FUNCTION_BLOCK FB_LeakTest
VAR_INPUT
    bExecute       		: BOOL;  		// Starts the leak test
    eSolenoidPosition 	: E_SolenoidSet;// Defines the solenoid valve positions
    tMonitorTime   		: TIME;  		// Monitoring time duration
    rPressureLimit 		: REAL;  		// Minimum required pressure limit
END_VAR

VAR_OUTPUT
    bLeakTestDone  : BOOL;  		// Indicates if the test was successful
    bLeakTestError : BOOL;  		// Indicates if an error occurred during the test
    sLTMessageError: STRING(100);  	// Error message describing the failure
END_VAR

VAR
    fbValveControl1 	: FB_ValvePositionControl;
    fbValveControl2 	: FB_ValvePositionControl;
    fbValveControl3 	: FB_ValvePositionControl;
    fbValveControl4 	: FB_ValvePositionControl;
    fbValveControl5 	: FB_ValvePositionControl;
    fbSolenoidControl 	: FB_SolenoidControl;
    fbSensorScale   	: FB_SensorScaling;
    tStartTime      	: TIME;
    rScaledPressure 	: REAL;
    eState          	: (IDLE, POSITION_VALVES, SET_SOLENOIDS, PRESSURIZE, MONITOR, DONE, ERROR);
END_VAR

CASE eState OF
    IDLE:
        // Waits for the execution command to start the test
        IF bExecute THEN
            eState := POSITION_VALVES;
        END_IF;

    POSITION_VALVES:
        // Moves all 6-position valves to position 5
        fbValveControl1(bEnable := TRUE, iValvePosition := 5, ServoAxis := GVL_Motion.M4Valve1.Axis);
        fbValveControl2(bEnable := TRUE, iValvePosition := 5, ServoAxis := GVL_Motion.M5Valve2.Axis);
        fbValveControl3(bEnable := TRUE, iValvePosition := 5, ServoAxis := GVL_Motion.M6Valve3.Axis);
        fbValveControl4(bEnable := TRUE, iValvePosition := 5, ServoAxis := GVL_Motion.M7Valve4.Axis);
        fbValveControl5(bEnable := TRUE, iValvePosition := 5, ServoAxis := GVL_Motion.M8Valve5.Axis);
        
        // If all valves have moved successfully, proceed to setting solenoids
        IF fbValveControl1.bMoveDone AND fbValveControl2.bMoveDone AND fbValveControl3.bMoveDone AND fbValveControl4.bMoveDone AND fbValveControl5.bMoveDone THEN
            eState := SET_SOLENOIDS;
        // If any valve encounters an error, transition to ERROR state
        ELSIF fbValveControl1.bError OR fbValveControl2.bError OR fbValveControl3.bError OR fbValveControl4.bError OR fbValveControl5.bError THEN
            bLeakTestError := TRUE;
            sLTMessageError := 'Failed to position valves';
            eState := ERROR;
        END_IF;
    
    SET_SOLENOIDS:
        // Sets the solenoids to LEAKTEST configuration
        fbSolenoidControl(bExecute := TRUE, eSolenoidSet := E_SolenoidSet.LEAKTEST);
        IF fbSolenoidControl.bDone THEN
            tStartTime := T#0S;
            eState := PRESSURIZE;
        END_IF;

    PRESSURIZE:
        // Waits for the pressurization time to complete
        tStartTime := tStartTime + T#1S;
        IF tStartTime >= tMonitorTime THEN
            // Switches solenoids to LEAKTESTMONITORING configuration before monitoring begins
            fbSolenoidControl(bExecute := TRUE, eSolenoidSet := E_SolenoidSet.LEAKTESTMONITORING);
            IF fbSolenoidControl.bDone THEN
                eState := MONITOR;
            END_IF;
        END_IF;

    MONITOR:
        // Reads and scales the pressure sensor value
        fbSensorScale(bExecute := TRUE, iRawValue := GVL_IO.gAnalogInputs.rMainPressureSupplyInput, iSensorID := 1, rPressure => rScaledPressure);
        
        // Verifies if the measured pressure meets the required limit
        IF rScaledPressure >= rPressureLimit THEN
            bLeakTestDone := TRUE;
            eState := DONE;
        ELSE
            bLeakTestError := TRUE;
            sLTMessageError := 'Pressure below required limit';
            eState := ERROR;
        END_IF;

    DONE:
        // Successfully completed the leak test
        bExecute := FALSE;

    ERROR:
        // Test encountered an error, execution halted
        bExecute := FALSE;
END_CASE;

END_FUNCTION_BLOCK

(* stored: Version 1.1.0.1, ProductVersion 3.1.4024.12
   POU FB_LeakTest: Id {21d6925c-1467-47b6-a1a0-80200f2aa3f7}, SpecialFunc None *)
